(* CODESYS project SingleResponsibility.project

Project tree, tasks and I/O mapping:
  Device : CODESYS Control Win V3, 3S - Smart Software Solutions GmbH, order no. 305021, version 3.5.10.40
    application Application
      libraries: Standard, * (System)
      task MainTask (cyclic, interval t#20ms, priority 1) calls PLC_PRG
      program PLC_PRG [ST]
  Basic/
    Sensor/
      interface ISensor: isOccupied, isFree
      function block DebouncedDigitalSensor [ST]: isOccupied, isFree, isRising, isFalling, FB_INIT, isSensorInState, updateState
    Edge/
      interface IEdge: isRising, isFalling
    Behaviour/
      interface IRunnable: run
      interface IStoppable: stop
      interface IEStoppable: executeEStop
  Conveyor/
    function block Conveyor2ndTry [ST]: run, FB_INIT, isEmpty, isAligned, isOccupiedInfeed, isOccupiedOutfeed
  Machine/
    interface IMachineState: isMachineInInitMode, isMachineInIdle, isMachineInSetup, isMachineInAutomatic, isMachineInEstop
  Drive/
    LinearDrive/
      interface ITwoStageLinearDrive: fastForward, forward, fastBackward, backward
    RotationalDrive/
      interface ITwoStageRotationDrive: fastClockwise, clockwise, fastCounterClockwise, counterClockwise
    function block ACommonTwoStageDrive [ST]: stop, fastForward, forward, fastBackward, backward, fastClockwise, clockwise, fastCounterClockwise, counterClockwise, executeEStop, FB_INIT
    function block Acme2StageDrive [ST]: stop, fastForward, forward, fastBackward, backward, fastClockwise, clockwise, fastCounterClockwise, counterClockwise, executeEStop, FB_INIT, StartMotor
  Communication/
    interface IReciverInterface: readExtCondition2Rec, isReceiving
    interface ISenderInterface: readExtCondition2Snd, isSending
    SMEMA/
      interface ISmema: setCondition, isTransferActive
      function block SmemaInterface [ST]: setCondition, isTransferActive, FB_INIT
      function block SmemaReceiver [ST]: isReceiving, readExtCondition2Rec, FB_INIT
      function block SmemaSender [ST]: readExtCondition2Snd, isSending, FB_INIT
*)

// Device/Application/PLC_PRG
PROGRAM PLC_PRG
VAR
END_VAR

END_PROGRAM

// Basic/Behaviour/IRunnable
INTERFACE IRunnable

METHOD run
VAR_INPUT
END_VAR
END_METHOD

END_INTERFACE

// Conveyor/Conveyor2ndTry
FUNCTION_BLOCK Conveyor2ndTry IMPLEMENTS IRunnable
VAR_INPUT
END_VAR
VAR_OUTPUT
END_VAR
VAR
	//sensors
	slowSensor			:ISensor; //sensor to slow down
	stopSensor			:ISensor; //sensor to stop
	//interfaces
	senderInterface		:ISenderInterface; //interface to send
	receiverInterface	:IReciverInterface; //interface to receive
	//conveyor drive
	drive 				:ITwoStageLinearDrive; //drive to run the conveyor
	//machine state
	machineState		:IMachineState; //just the machine state
END_VAR

METHOD run
(*recive part*)
	IF (THIS^.receiverInterface.readExtCondition2Rec(receiveCondition := THIS^.isEmpty()).isReceiving()) THEN
		THIS^.drive.fastForward();
	(*send part*)
	ELSIF (THIS^.senderInterface.readExtCondition2Snd(sendCondition := (THIS^.isAligned() OR THIS^.isOccupiedOutfeed())).isSending()) THEN
		THIS^.drive.fastForward();
	(*align part*)
	ELSIF (THIS^.isOccupiedInfeed() AND THIS^.machineState.isMachineInAutomatic()) THEN
		THIS^.drive.forward();
	ELSE
		THIS^.drive.stop();
	END_IF
END_METHOD

METHOD FB_INIT
VAR_INPUT
	//CODESYS stuff
	bInitRetains		:BOOL; // initializing of retain-variable
	bInCopyCode 		:BOOL; // instance is copied to copy-code
	//sensors
	slowSensor			:ISensor; //sensor to slow down
	stopSensor			:ISensor; //sensor to stop
	//interfaces
	senderInterface		:ISenderInterface; //interface to send
	receiverInterface	:IReciverInterface; //interface to receive
	//conveyor drive
	drive 				:ITwoStageLinearDrive; //drive to run the conveyor
	//machine state
	machineState		:IMachineState; //just the machine state
END_VAR
//sensors
THIS^.slowSensor	    := slowSensor; //sensor to slow down
THIS^.stopSensor	    := stopSensor; //sensor to stop
//interfaces
THIS^.senderInterface	:= senderInterface	; //interface to send
THIS^.receiverInterface	:= receiverInterface; //interface to receive
//conveyor drive
THIS^.drive 			:= drive; //drive to run the conveyor
//machine state
THIS^.machineState		:= machineState; //just the machine state
END_METHOD

METHOD isEmpty : BOOL
VAR_INPUT
END_VAR
isEmpty := (THIS^.slowSensor.isFree() AND THIS^.stopSensor.isFree());
END_METHOD

METHOD isAligned : BOOL
VAR_INPUT
END_VAR
isAligned := (THIS^.slowSensor.isOccupied() AND THIS^.stopSensor.isOccupied());
END_METHOD

METHOD isOccupiedInfeed : BOOL
VAR_INPUT
END_VAR
isOccupiedInfeed := (THIS^.slowSensor.isOccupied() AND THIS^.stopSensor.isFree());
END_METHOD

METHOD isOccupiedOutfeed : BOOL
VAR_INPUT
END_VAR
isOccupiedOutfeed := (THIS^.slowSensor.isFree() AND THIS^.stopSensor.isOccupied());
END_METHOD

END_FUNCTION_BLOCK

// Basic/Sensor/ISensor
INTERFACE ISensor

METHOD isOccupied : BOOL
VAR_INPUT
END_VAR
END_METHOD

METHOD isFree : BOOL
VAR_INPUT
END_VAR
END_METHOD

END_INTERFACE

// Communication/ISenderInterface
INTERFACE ISenderInterface

(*inject conditions for ready to receive*)
METHOD readExtCondition2Snd : ISenderInterface
VAR_INPUT
	sendCondition	:BOOL; //condition 4 ready 2 send
END_VAR
VAR
	
END_VAR
END_METHOD

METHOD isSending : BOOL
VAR_INPUT
END_VAR
END_METHOD

END_INTERFACE

// Communication/IReciverInterface
INTERFACE IReciverInterface

(*inject conditions for ready to receive*)
METHOD readExtCondition2Rec : IReciverInterface
VAR_INPUT
	receiveCondition	:BOOL; //condition 4 ready to receive
END_VAR
VAR 
END_VAR
END_METHOD

METHOD isReceiving : BOOL
VAR_INPUT
END_VAR
END_METHOD

END_INTERFACE

// Drive/LinearDrive/ITwoStageLinearDrive
INTERFACE ITwoStageLinearDrive EXTENDS IStoppable

METHOD fastForward
VAR_INPUT
END_VAR
END_METHOD

METHOD forward
VAR_INPUT
END_VAR
END_METHOD

METHOD fastBackward
VAR_INPUT
END_VAR
END_METHOD

METHOD backward
VAR_INPUT
END_VAR
END_METHOD

END_INTERFACE

// Basic/Behaviour/IStoppable
INTERFACE IStoppable

METHOD stop
VAR_INPUT
END_VAR
END_METHOD

END_INTERFACE

// Machine/IMachineState
INTERFACE IMachineState

(*Init mode for first init cycle during start-up*)
METHOD isMachineInInitMode : BOOL
VAR_INPUT
END_VAR
END_METHOD

(*Idle means machine is ready to change to setup or automatic mode*)
METHOD isMachineInIdle : BOOL
VAR_INPUT
END_VAR
END_METHOD

(*setup is for manually operated actions*)
METHOD isMachineInSetup : BOOL
VAR_INPUT
END_VAR
END_METHOD

(*automatic means machine is running in production*)
METHOD isMachineInAutomatic : BOOL
VAR_INPUT
END_VAR
END_METHOD

(*e-stop means machine is in e-stop*)
METHOD isMachineInEstop : BOOL
VAR_INPUT
END_VAR
END_METHOD

END_INTERFACE

// Basic/Edge/IEdge
INTERFACE IEdge

METHOD isRising : BOOL
VAR_INPUT
END_VAR
END_METHOD

METHOD isFalling : BOOL
VAR_INPUT
END_VAR
END_METHOD

END_INTERFACE

// Basic/Behaviour/IEStoppable
INTERFACE IEStoppable

METHOD executeEStop
VAR_INPUT
END_VAR
END_METHOD

END_INTERFACE

// Drive/RotationalDrive/ITwoStageRotationDrive
INTERFACE ITwoStageRotationDrive EXTENDS IStoppable

METHOD fastClockwise
VAR_INPUT
END_VAR
END_METHOD

METHOD clockwise
VAR_INPUT
END_VAR
END_METHOD

METHOD fastCounterClockwise
VAR_INPUT
END_VAR
END_METHOD

METHOD counterClockwise
VAR_INPUT
END_VAR
END_METHOD

END_INTERFACE

// Drive/ACommonTwoStageDrive
{info 'ACommonTwoStageDrive is just an abstract class'}
FUNCTION_BLOCK ACommonTwoStageDrive IMPLEMENTS ITwoStageLinearDrive, ITwoStageRotationDrive, IEStoppable
VAR_INPUT
END_VAR
VAR_OUTPUT
END_VAR
VAR
END_VAR

METHOD stop
END_METHOD

METHOD fastForward
END_METHOD

METHOD forward
END_METHOD

METHOD fastBackward
END_METHOD

METHOD backward
END_METHOD

METHOD fastClockwise
END_METHOD

METHOD clockwise
END_METHOD

METHOD fastCounterClockwise
END_METHOD

METHOD counterClockwise
END_METHOD

METHOD executeEStop
END_METHOD

METHOD FB_INIT
VAR_INPUT
	//CODESYS stuff
	bInitRetains	:BOOL; // initializing of retain-variable
	bInCopyCode 	:BOOL; // instance is copied to copy-code
END_VAR
END_METHOD

END_FUNCTION_BLOCK

// Drive/Acme2StageDrive
FUNCTION_BLOCK Acme2StageDrive EXTENDS ACommonTwoStageDrive
VAR_INPUT
END_VAR
VAR_OUTPUT
END_VAR
VAR
	//drive signals
	cw				:REFERENCE TO BOOL; //run the motor clockwise, if it false the motor will run counter clockwise
	fast			:REFERENCE TO BOOL; //run the motor fast, if it false will the motor running slow
	start			:REFERENCE TO BOOL; //run start the motor
	maskFwd			:BOOL; //mask to define forward or rather clockwise
END_VAR

METHOD stop
THIS^.start := FALSE;
END_METHOD

METHOD fastForward
THIS^.StartMotor(direction := THIS^.maskFwd, velocity := TRUE);
END_METHOD

METHOD forward
THIS^.StartMotor(direction := THIS^.maskFwd, velocity := FALSE);
END_METHOD

METHOD fastBackward
THIS^.StartMotor(direction := (NOT THIS^.maskFwd), velocity := TRUE);
END_METHOD

METHOD backward
THIS^.StartMotor(direction := (NOT THIS^.maskFwd), velocity := FALSE);
END_METHOD

METHOD fastClockwise
THIS^.fastForward();
END_METHOD

METHOD clockwise
THIS^.forward();
END_METHOD

METHOD fastCounterClockwise
THIS^.fastBackward();
END_METHOD

METHOD counterClockwise
THIS^.backward();
END_METHOD

METHOD executeEStop
THIS^.stop();
END_METHOD

METHOD FB_INIT
VAR_INPUT
	//CODESYS stuff
	bInitRetains	:BOOL; // initializing of retain-variable
	bInCopyCode 	:BOOL; // instance is copied to copy-code
	//drive signals
	cw				:REFERENCE TO BOOL; //run the motor clockwise, if it false the motor will run counter clockwise
	fast			:REFERENCE TO BOOL; //run the motor fast, if it false will the motor running slow
	start			:REFERENCE TO BOOL; //run start the motor
	maskFwd			:BOOL; //mask to define forward or rather clockwise
END_VAR
THIS^.cw             REF= cw ;
THIS^.fast           REF= fast ;
THIS^.start          REF= start ;
THIS^.maskFwd      	 :=   maskFwd;
END_METHOD

METHOD PROTECTED StartMotor
VAR_INPUT
	direction :BOOL; //direction flag
	velocity: BOOL; //velocity flag
END_VAR
THIS^.cw 	 	:= direction;
THIS^.fast   	:= velocity;
THIS^.start  	:= TRUE;
END_METHOD

END_FUNCTION_BLOCK

// Basic/Sensor/DebouncedDigitalSensor
FUNCTION_BLOCK DebouncedDigitalSensor IMPLEMENTS ISensor, IEdge
VAR_INPUT
END_VAR
VAR_OUTPUT
END_VAR
VAR
	diSensor			:REFERENCE TO BOOL; //reference to the digital input
	maskOccupied		:BOOL; //mask for the state occupied
	debouncer			:TON; //ton to debounce the sensor signal
	debounceTime		:TIME; //debounce time
	state				:BOOL; //sensor state 
END_VAR

METHOD isOccupied : BOOL
isOccupied := isSensorInState(state := THIS^.maskOccupied);
END_METHOD

METHOD isFree : BOOL
isFree := isSensorInState(state := (NOT THIS^.maskOccupied));
END_METHOD

METHOD isRising : BOOL
isRising 	:= (THIS^.isOccupied() AND (NOT THIS^.state));
THIS^.updateState();
END_METHOD

METHOD isFalling : BOOL
isFalling 	:= (THIS^.isFree() AND THIS^.state);
THIS^.updateState();
END_METHOD

METHOD FB_INIT
VAR_INPUT
	//CODESYS stuff
	bInitRetains	:BOOL; // initializing of retain-variable
	bInCopyCode 	:BOOL; // instance is copied to copy-code
	//the sensor
	diSensor		:REFERENCE TO BOOL; //reference to the digital input
	maskOccupied	:BOOL; //mask for the state occupied
END_VAR
THIS^.diSensor		REF=diSensor; 
THIS^.maskOccupied	:= maskOccupied;
THIS^.debounceTime	:= T#30ms;
THIS^.state			:= (THIS^.diSensor = THIS^.maskOccupied);
END_METHOD

METHOD PROTECTED isSensorInState : BOOL
VAR_INPUT
	state :BOOL; //requeseted sensor state
END_VAR
THIS^.debouncer(IN := (THIS^.diSensor = state), PT := THIS^.debounceTime, Q => isSensorInState);
END_METHOD

METHOD PROTECTED updateState
VAR_INPUT
END_VAR
THIS^.state := THIS^.isOccupied();
END_METHOD

END_FUNCTION_BLOCK

// Communication/SMEMA/ISmema
INTERFACE ISmema

METHOD setCondition
VAR_INPUT
	smemaCondition	:BOOL; //must be ture to activate the smema interface
END_VAR
END_METHOD

METHOD isTransferActive : BOOL
VAR_INPUT
END_VAR
END_METHOD

END_INTERFACE

// Communication/SMEMA/SmemaInterface
FUNCTION_BLOCK SmemaInterface IMPLEMENTS ISmema
VAR_INPUT
END_VAR
VAR_OUTPUT
END_VAR
VAR
	machineStateHndl	:IMachineState; //machine state handler to check if receiving is allowed
	partnerIsRdy	    :REFERENCE TO BOOL; //ready signal from the interface partner
	weAreRdy			:REFERENCE TO BOOL; //ready signal to the interface partner
	transferCondition	:BOOL; //external condition for transfer is possible
	maskPartnerIsRdy	:BOOL; //bitmask for partner is ready
	maskWeAreRdy		:BOOL; //bitmask for we are ready	

END_VAR

METHOD setCondition
VAR_INPUT
	(*must be ture to activate the smema interface*)
	smemaCondition	: BOOL;
END_VAR
THIS^.transferCondition	:= transferCondition;
IF (NOT THIS^.transferCondition) THEN
	THIS^.weAreRdy := (NOT THIS^.maskWeAreRdy);
END_IF;
END_METHOD

METHOD isTransferActive : BOOL
IF (THIS^.transferCondition AND THIS^.machineStateHndl.isMachineInAutomatic()) THEN
	THIS^.weAreRdy := THIS^.maskWeAreRdy;
ELSE
	THIS^.weAreRdy := (NOT THIS^.maskWeAreRdy);
END_IF;		
isTransferActive	  := ((THIS^.weAreRdy = THIS^.maskWeAreRdy) AND (THIS^.maskPartnerIsRdy = THIS^.maskPartnerIsRdy));
END_METHOD

METHOD FB_INIT
VAR_INPUT
	//CODESYS stuff
	bInitRetains			:BOOL; // initializing of retain-variable
	bInCopyCode 			:BOOL; // instance is copied to copy-code
	//interface signals
	partnerIsRdy	        :REFERENCE TO BOOL; //ready signal from the interface partner
	weAreRdy			    :REFERENCE TO BOOL; //ready signal to the interface partner
	//bit masks
	maskPartnerIsRdy		:BOOL; //bitmask for partner is ready
	maskWeAreRdy			:BOOL; //bitmask for we are ready	
	//machine state
	machineStateHndl		:IMachineState; //the machine is in machine state automatic
END_VAR
THIS^.partnerIsRdy	    REF= partnerIsRdy;
THIS^.weAreRdy		    REF= weAreRdy;
THIS^.machineStateHndl	:= 	 machineStateHndl;
THIS^.transferCondition	:=	 FALSE;
THIS^.maskPartnerIsRdy	:=   maskPartnerIsRdy;
THIS^.maskWeAreRdy		:=	 maskWeAreRdy;
END_METHOD

END_FUNCTION_BLOCK

// Communication/SMEMA/SmemaReceiver
FUNCTION_BLOCK SmemaReceiver IMPLEMENTS IReciverInterface
VAR_INPUT
END_VAR
VAR_OUTPUT
END_VAR
VAR
	smeaInterface :ISmema; //smema interface for the receiver
END_VAR

METHOD isReceiving : BOOL
isReceiving	  := (THIS^.smeaInterface.isTransferActive());
END_METHOD

(*inject conditions for ready to receive*)
METHOD readExtCondition2Rec : IReciverInterface
VAR_INPUT
	receiveCondition	:BOOL; //condition 4 ready to receive
END_VAR
VAR 
	
END_VAR
THIS^.smeaInterface.setCondition(smemaCondition := receiveCondition);
readExtCondition2Rec	:= THIS^;
END_METHOD

METHOD FB_INIT
VAR_INPUT
	//CODESYS stuff
	bInitRetains			:BOOL; // initializing of retain-variable
	bInCopyCode 			:BOOL; // instance is copied to copy-code
	//smems interface
	smeaInterface :ISmema; //smema interface for the receiver
END_VAR
THIS^.smeaInterface	:= 	 smeaInterface ;
END_METHOD

END_FUNCTION_BLOCK

// Communication/SMEMA/SmemaSender
FUNCTION_BLOCK SmemaSender IMPLEMENTS ISenderInterface
VAR_INPUT
END_VAR
VAR_OUTPUT
END_VAR
VAR
	smeaInterface :ISmema; //smema interface for the sender
END_VAR

(*inject conditions for ready to receive*)
METHOD readExtCondition2Snd : ISenderInterface
VAR_INPUT
	sendCondition	:BOOL; //condition 4 ready 2 send
END_VAR
VAR
	
END_VAR
THIS^.smeaInterface.setCondition(smemaCondition := sendCondition);
readExtCondition2Snd := THIS^;
END_METHOD

METHOD isSending : BOOL
isSending	  := (THIS^.smeaInterface.isTransferActive());
END_METHOD

METHOD FB_INIT
VAR_INPUT
	//CODESYS stuff
	bInitRetains			:BOOL; // initializing of retain-variable
	bInCopyCode 			:BOOL; // instance is copied to copy-code
	//smems interface
	smeaInterface :ISmema; //smema interface for the sender
END_VAR
THIS^.smeaInterface	:= 	 smeaInterface ;
END_METHOD

END_FUNCTION_BLOCK
